TYPE E_ComState :
(
	INIT := 0,
	IDLE,
	CONNECT,
	DATATRANSFER,
	DISCONNECT
);
END_TYPE

(* stored: Version 1.1.0.1, ProductVersion 3.1.4024.6
   DUT E_ComState: Id {d4be720f-11f2-4cb9-9d95-eece16bad425} *)
